// TIA Portal V20 export
FUNCTION_BLOCK "FB_Read_Data_SR-X100W"   // FB6, LAD
{ S7_Optimized_Access := 'TRUE' }
// stored: AutoNumber false, MemoryReserve 100, SetENOAutomatically false
   VAR_INPUT
      Trigger_Sensor : Bool;
      Read_Complete : Bool;
      Read_Failure : Bool;
      Clear_Data : Bool;
      Read_Data_In : "SR-X100W_Read_Data";
   END_VAR
   VAR_OUTPUT
      Read_Request : Bool;
      Read_Complete_Clear : Bool;
      Read_Complete_OUT : Bool;
      Read_Failure_OUT : Bool;
      Read_Data_Out : String[136];
      Serial_Number { ExternalAccessible := 'False'; ExternalVisible := 'False'; ExternalWritable := 'False'} : String[17];
   END_VAR
   VAR
      Aux_Triggger_1 : Bool;
      Aux_Triggger_2 : Bool;
      Aux_Triggger_3 : Bool;
      Aux_Triggger_4 : Bool;
      DB_What_Was_Read_Instance { S7_SetPoint := 'True'} : "FB_What_Was_Read";
      Timer_Delay_Reset { S7_SetPoint := 'True'} : TON_TIME;
   END_VAR
   VAR_TEMP   // added for the SCL form of the ladder/FBD networks
      _w1 : Bool;
      _w2 : Bool;
   END_VAR
BEGIN

REGION Network 1
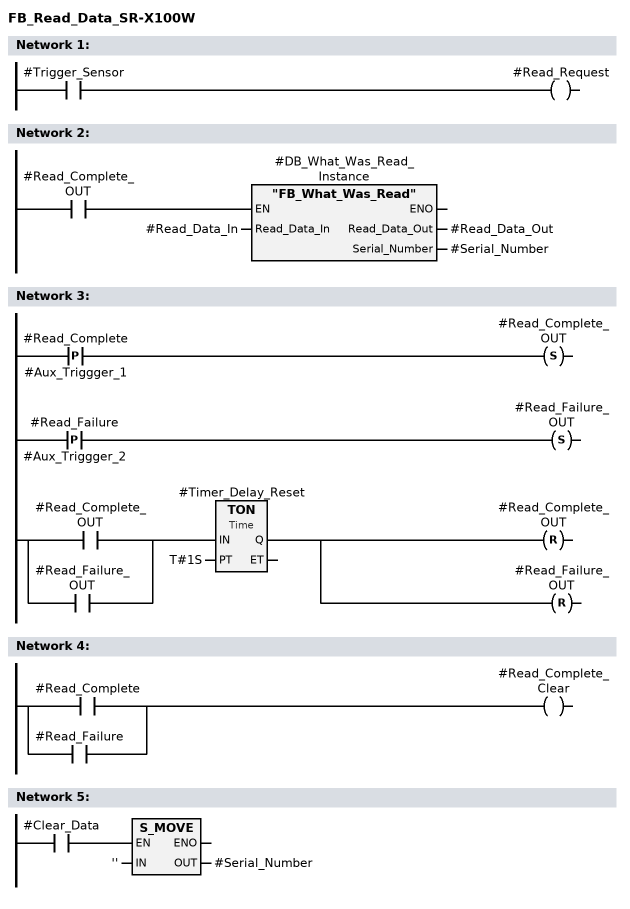
   RUNG wire#powerrail
      Contact( #Trigger_Sensor )
      Coil( #Read_Request )
   END_RUNG
   // the same network as SCL:
   #Read_Request := #Trigger_Sensor;
END_REGION

REGION Network 2
   RUNG wire#powerrail
      Contact( #Read_Complete_OUT )
      #DB_What_Was_Read_Instance(Read_Data_In := #Read_Data_In, Read_Data_Out => #Read_Data_Out, Serial_Number => #Serial_Number)
   END_RUNG
   // the same network as SCL:
   IF #Read_Complete_OUT THEN
       #DB_What_Was_Read_Instance(Read_Data_In := #Read_Data_In,   // "FB_What_Was_Read"
                               Read_Data_Out => #Read_Data_Out,
                               Serial_Number => #Serial_Number);
   END_IF;
END_REGION

REGION Network 3
   RUNG wire#powerrail
      P_Contact(operand := #Read_Complete, bit := #Aux_Triggger_1)
      S_Coil( #Read_Complete_OUT )
   END_RUNG
   RUNG wire#powerrail
      P_Contact(operand := #Read_Failure, bit := #Aux_Triggger_2)
      S_Coil( #Read_Failure_OUT )
   END_RUNG
   RUNG wire#powerrail
      Contact( #Read_Complete_OUT )
      wire#w1
      { S7_Templates := "time_type := Time" } #Timer_Delay_Reset.TON(pt := T#1S, et =>)
      wire#w2
      R_Coil( #Read_Complete_OUT )
   END_RUNG
   RUNG wire#powerrail
      Contact( #Read_Failure_OUT )
   END_RUNG wire#w1
   RUNG wire#w2
      R_Coil( #Read_Failure_OUT )
   END_RUNG
   // the same network as SCL:
   #_w1 := #Read_Complete AND NOT #Aux_Triggger_1;   // rising edge of #Read_Complete
   #Aux_Triggger_1 := #Read_Complete;
   IF #_w1 THEN #Read_Complete_OUT := TRUE; END_IF;
   #_w2 := #Read_Failure AND NOT #Aux_Triggger_2;   // rising edge of #Read_Failure
   #Aux_Triggger_2 := #Read_Failure;
   IF #_w2 THEN #Read_Failure_OUT := TRUE; END_IF;
   #Timer_Delay_Reset(IN := #Read_Complete_OUT OR #Read_Failure_OUT, PT := T#1S);   // TON
   IF #Timer_Delay_Reset.Q THEN
       #Read_Complete_OUT := FALSE;
       #Read_Failure_OUT := FALSE;
   END_IF;
END_REGION

REGION Network 4
   RUNG wire#powerrail
      Contact( #Read_Complete )
      wire#w1
      Coil( #Read_Complete_Clear )
   END_RUNG
   RUNG wire#powerrail
      Contact( #Read_Failure )
   END_RUNG wire#w1
   // the same network as SCL:
   #Read_Complete_Clear := #Read_Complete OR #Read_Failure;
END_REGION

REGION Network 5
   RUNG wire#powerrail
      Contact( #Clear_Data )
      S_Move(in := '', out => #Serial_Number)
   END_RUNG
   // the same network as SCL:
   IF #Clear_Data THEN #Serial_Number := ''; END_IF;
END_REGION
END_FUNCTION_BLOCK
